# B&R Automation Studio project TD52 (part 12)

### blascompat32.h
```c
/*
 * @(#)blascompat32.h    generated by: makeheader 5.1.5  Tue May 24 21:10:38 2011
 *
 *		built from:	../../src/include/copyright.h
 *				../../src/include/pragma_interface.h
 *				include/blascompat32/blascompat32.h
 */

#if defined(_MSC_VER)
# pragma once
#endif
#if defined(__GNUC__) && (__GNUC__ > 3 || (__GNUC__ == 3 && __GNUC_MINOR__ > 3))
# pragma once
#endif

#ifndef blascompat32_h
#define blascompat32_h

/*
 * Copyright 1984-2003 The MathWorks, Inc.
 * All Rights Reserved.
 */

/* Copyright 2003-2006 The MathWorks, Inc. */

/* Only define EXTERN_C if it hasn't been defined already. This allows
 * individual modules to have more control over managing their exports.
 */
#ifndef EXTERN_C

#ifdef __cplusplus
  #define EXTERN_C extern "C"
#else
  #define EXTERN_C extern
#endif

#endif

/*
 * CONFIDENTIAL AND CONTAINING PROPRIETARY TRADE SECRETS
 * Copyright 1984-2009 The MathWorks, Inc.
 * The source code contained in this listing contains proprietary and
 * confidential trade secrets of The MathWorks, Inc.   The use, modification,
 * or development of derivative work based on the code or ideas obtained
 * from the code is prohibited without the express written permission of The
 * MathWorks, Inc.  The disclosure of this code to any party not authorized
 * by The MathWorks, Inc. is strictly forbidden.
 * CONFIDENTIAL AND CONTAINING PROPRIETARY TRADE SECRETS
 */

/*
   32-bit API wrapper for libmwblas
   WARNING: This module is a temporary module specifically designed to
            bridge the incompatiblity between Embedded MATLAB (which lacks
            a 64-bit integer type) and 64-bit BLAS only.
            Do not link to this module otherwise.
            Link to libmwblas instead.
 */
#include <tmwtypes.h>

#if defined(_WIN32)
#define FORTRAN_WRAPPER(x) x
#else
#define FORTRAN_WRAPPER(x) x ## _
#endif

#ifndef COMPLEX_TYPES
#define COMPLEX_TYPES
  typedef struct{float r,i;} complex;
  typedef struct{double r,i;} doublecomplex;
#endif

#define isamax32 FORTRAN_WRAPPER(isamax32)
EXTERN_C int isamax32(const int *n32, const float  *sx, const int *incx32);

#define idamax32 FORTRAN_WRAPPER(idamax32)
EXTERN_C int idamax32(const int *n32, const double *dx, const int *incx32);

#define icamax32 FORTRAN_WRAPPER(icamax32)
EXTERN_C int icamax32(const int *n32, const creal32_T *cx, const int *incx32);

#define izamax32 FORTRAN_WRAPPER(izamax32)
EXTERN_C int izamax32(const int *n32, const creal_T *zx, const int *incx32);

#define sasum32 FORTRAN_WRAPPER(sasum32)
EXTERN_C float sasum32(const int *n32, const float  *sx, const int *incx32);

#define dasum32 FORTRAN_WRAPPER(dasum32)
EXTERN_C double dasum32(const int *n32, const double *dx, const int *incx32);

#define saxpy32 FORTRAN_WRAPPER(saxpy32)
EXTERN_C void saxpy32(const int *n32, const float *sa, const float  *sx,
             const int *incx32, float *sy, const int *incy32);

#define daxpy32 FORTRAN_WRAPPER(daxpy32)
EXTERN_C void daxpy32(const int *n32, const double *da, const double *dx,
             const int *incx32, double *dy, const int *incy32);

#define caxpy32 FORTRAN_WRAPPER(caxpy32)
EXTERN_C void caxpy32(const int *n32, const creal32_T *ca, const creal32_T *cx,
             const int *incx32, creal32_T *cy, const int *incy32);

#define zaxpy32 FORTRAN_WRAPPER(zaxpy32)
EXTERN_C void zaxpy32(const int *n32, const creal_T *za, const creal_T *zx,
             const int *incx32, creal_T *zy, const int *incy32);

#define scopy32 FORTRAN_WRAPPER(scopy32)
EXTERN_C void scopy32(const int *n32, const float *sx, const int *incx32,
             float *sy, const int *incy32);

#define dcopy32 FORTRAN_WRAPPER(dcopy32)
EXTERN_C void dcopy32(const int *n32, const double *dx, const int *incx32,
             double *dy, const int *incy32);

#define ccopy32 FORTRAN_WRAPPER(ccopy32)
EXTERN_C void ccopy32(const int *n32, const creal32_T *cx, const int *incx32,
             creal32_T *cy, const int *incy32);

#define zcopy32 FORTRAN_WRAPPER(zcopy32)
EXTERN_C void zcopy32(const int *n32, creal_T *zx, const int *incx32,
             creal_T *zy, const int *incy32);

#define cdotc32 FORTRAN_WRAPPER(cdotc32)
EXTERN_C complex cdotc32(const int *n32, const creal32_T *cx, const int *incx32,
              const creal32_T *cy, const int *incy32);

#define zdotc32 FORTRAN_WRAPPER(zdotc32)
EXTERN_C doublecomplex zdotc32(const int *n32, const creal_T *zx, const int *incx32,
               const creal_T *zy, const int *incy32);

#define sdot32 FORTRAN_WRAPPER(sdot32)
EXTERN_C float sdot32(const int *n32, const float *sx, const int *incx32,
             const float  *sy, const int *incy32);

#define ddot32 FORTRAN_WRAPPER(ddot32)
EXTERN_C double ddot32(const int *n32, const double *dx, const int *incx32,
              const double *dy, const int *incy32);

#define cdotu32 FORTRAN_WRAPPER(cdotu32)
EXTERN_C complex cdotu32(const int *n32, const creal32_T *cx, const int *incx32,
              const creal32_T *cy, const int *incy32);

#define zdotu32 FORTRAN_WRAPPER(zdotu32)
EXTERN_C doublecomplex zdotu32(const int *n32, const creal_T *zx, const int *incx32,
               const creal_T *zy, const int *incy32);

#define sgemm32 FORTRAN_WRAPPER(sgemm32)
EXTERN_C void sgemm32(char *transa, char *transb, const int *m32, const int *n32,
             const int *k32, const float *alpha, const float *a, const int *lda32,
             const float *b, const int *ldb32, const float *beta, float *c,
             const int *ldc32);

#define dgemm32 FORTRAN_WRAPPER(dgemm32)
EXTERN_C void dgemm32(char *transa, char *transb, const int *m32, const int *n32,
             const int *k32, const double *alpha, const double *a, const int *lda32,
             const double *b, const int *ldb32, const double *beta, double  *c,
             const int *ldc32);

#define cgemm32 FORTRAN_WRAPPER(cgemm32)
EXTERN_C void cgemm32(char *transa, char *transb, const int *m32, const int *n32,
             const int *k32, const creal32_T *alpha, const creal32_T *a, const int *lda32,
             const creal32_T *b, const int *ldb32, const creal32_T *beta, creal32_T *c,
             const int *ldc32);

#define zgemm32 FORTRAN_WRAPPER(zgemm32)
EXTERN_C void zgemm32(char *transa, char *transb, const int *m32, const int *n32,
             const int *k32, const creal_T *alpha, const creal_T *a, const int *lda32,
             const creal_T *b, const int *ldb32, const creal_T *beta, creal_T *c,
             const int *ldc32);

#define sgemv32 FORTRAN_WRAPPER(sgemv32)
EXTERN_C void sgemv32(char *trans, const int *m32, const int *n32, const float *alpha,
             const float *a, const int *lda32, const float *x, const int *incx32,
             const float *beta, float *y, const int *incy32);

#define dgemv32 FORTRAN_WRAPPER(dgemv32)
EXTERN_C void dgemv32(char *trans, const int *m32, const int *n32, const double *alpha,
             const double *a, const int *lda32, const double *x, const int *incx32,
             const double *beta, double *y, const int *incy32);

#define cgemv32 FORTRAN_WRAPPER(cgemv32)
EXTERN_C void cgemv32(char *trans, const int *m32, const int *n32, const creal32_T *alpha,
             const creal32_T *a, const int *lda32, const creal32_T *x, const int *incx32,
             const creal32_T *beta, creal32_T *y, const int *incy32);

#define zgemv32 FORTRAN_WRAPPER(zgemv32)
EXTERN_C void zgemv32(char *trans, const int *m32, const int *n32, const creal_T *alpha,
             const creal_T *a, const int *lda32, const creal_T *x, const int *incx32,
             const creal_T *beta, creal_T *y, const int *incy32);

#define cgerc32 FORTRAN_WRAPPER(cgerc32)
EXTERN_C void cgerc32(const int *m32, const int *n32, const creal32_T *alpha, const creal32_T *x,
             const int *incx32, const creal32_T *y, const int *incy32,
             creal32_T *a, const int *lda32);

#define zgerc32 FORTRAN_WRAPPER(zgerc32)
EXTERN_C void zgerc32(const int *m32, const int *n32, const creal_T *alpha, const creal_T *x,
             const int *incx32, creal_T *y, const int *incy32,
             creal_T *a, const int *lda32);

#define sger32 FORTRAN_WRAPPER(sger32)
EXTERN_C void sger32(const int *m32, const int *n32, const float *alpha, const float  *x,
            const int *incx32, const float *y, const int *incy32,
            float *a, const int *lda32);

#define dger32 FORTRAN_WRAPPER(dger32)
EXTERN_C void dger32(const int *m32, const int *n32, const double *alpha, const double *x,
            const int *incx32, const double *y, const int *incy32,
            double *a, const int *lda32);

#define cgeru32 FORTRAN_WRAPPER(cgeru32)
EXTERN_C void cgeru32(const int *m32, const int *n32, const creal32_T *alpha, const creal32_T *x,
             const int *incx32, const creal32_T *y, const int *incy32,
             creal32_T *a, const int *lda32);

#define zgeru32 FORTRAN_WRAPPER(zgeru32)
EXTERN_C void zgeru32(const int *m32, const int *n32, const creal_T *alpha, const creal_T *x,
             const int *incx32, creal_T *y, const int *incy32,
             creal_T *a, const int *lda32);

#define snrm232 FORTRAN_WRAPPER(snrm232)
EXTERN_C float snrm232(const int *n32, const float *x, const int *incx32);

#define dnrm232 FORTRAN_WRAPPER(dnrm232)
EXTERN_C double dnrm232(const int *n32, const double *x, const int *incx32);

#define scnrm232 FORTRAN_WRAPPER(scnrm232)
EXTERN_C float scnrm232(const int *n32, const creal32_T *x, const int *incx32);

#define dznrm232 FORTRAN_WRAPPER(dznrm232)
EXTERN_C double dznrm232(const int *n32, const creal_T *x, const int *incx32);

#define srotg32 FORTRAN_WRAPPER(srotg32)
EXTERN_C void srotg32(float  *sa, float  *sb, float  *c, float  *s);

#define drotg32 FORTRAN_WRAPPER(drotg32)
EXTERN_C void drotg32(double *da, double *db, double *c, double *s);

#define crotg32 FORTRAN_WRAPPER(crotg32)
EXTERN_C void crotg32(creal32_T *ca, creal32_T *cb, creal32_T *c, creal32_T *s);

#define zrotg32 FORTRAN_WRAPPER(zrotg32)
EXTERN_C void zrotg32(creal_T *ca, creal_T *cb, creal_T *c, creal_T *s);

#define srot32 FORTRAN_WRAPPER(srot32)
EXTERN_C void srot32(const int *n32, float  *sx, const int *incx32, float  *sy,
            const int *incy32, const float *c, const float *s);

#define drot32 FORTRAN_WRAPPER(drot32)
EXTERN_C void drot32(const int *n32, double *dx, const int *incx32, double *dy,
            const int *incy32, const double *c, const double *s);

#define csrot32 FORTRAN_WRAPPER(csrot32)
EXTERN_C void csrot32(const int *n32, creal32_T *cx, const int *incx32, creal32_T *cy,
             const int *incy32, const float *c, const creal32_T *s);

#define zdrot32 FORTRAN_WRAPPER(zdrot32)
EXTERN_C void zdrot32(const int *n32, creal_T *cx, const int *incx32, creal_T *cy,
             const int *incy32, const double *c, const creal_T *s);

#define sscal32 FORTRAN_WRAPPER(sscal32)
EXTERN_C void sscal32(const int *n32, const float *sa, float  *sx, const int *incx32);

#define dscal32 FORTRAN_WRAPPER(dscal32)
EXTERN_C void dscal32(const int *n32, const double *da, double *dx, const int *incx32);

#define cscal32 FORTRAN_WRAPPER(cscal32)
EXTERN_C void cscal32(const int *n32, const creal32_T *ca, creal32_T *cx, const int *incx32);

#define zscal32 FORTRAN_WRAPPER(zscal32)
EXTERN_C void zscal32(const int *n32, const creal_T *za, creal_T *zx, const int *incx32);

#define sswap32 FORTRAN_WRAPPER(sswap32)
EXTERN_C void sswap32(const int *n32, float  *sx, const int *incx32, float  *sy,
             const int *incy32);

#define dswap32 FORTRAN_WRAPPER(dswap32)
EXTERN_C void dswap32(const int *n32, double *dx, const int *incx32, double *dy,
             const int *incy32);

#define cswap32 FORTRAN_WRAPPER(cswap32)
EXTERN_C void cswap32(const int *n32, creal32_T *cx, const int *incx32,
             creal32_T *cy, const int *incy32);

#define zswap32 FORTRAN_WRAPPER(zswap32)
EXTERN_C void zswap32(const int *n32, creal_T *zx, const int *incx32,
             creal_T *zy, const int *incy32);

#define strsm32 FORTRAN_WRAPPER(strsm32)
EXTERN_C void strsm32(char   *side, char   *uplo, char   *transa,
             char *diag, const int *m32, const int *n32,
             const float *alpha, const float *a, const int *lda32,
             float  *b, const int *ldb32);

#define dtrsm32 FORTRAN_WRAPPER(dtrsm32)
EXTERN_C void dtrsm32(char   *side, char   *uplo, char   *transa,
             char *diag, const int *m32, const int *n32,
             const double *alpha, const double *a, const int *lda32,
             double *b, const int *ldb32);

#define ctrsm32 FORTRAN_WRAPPER(ctrsm32)
EXTERN_C void ctrsm32(char   *side, char   *uplo, char   *transa,
             char *diag, const int *m32, const int *n32,
             const creal32_T *alpha, const creal32_T *a, const int *lda32,
             creal32_T *b, const int *ldb32);

#define ztrsm32 FORTRAN_WRAPPER(ztrsm32)
EXTERN_C void ztrsm32(char   *side, char   *uplo, char   *transa,
             char *diag, const int *m32, const int *n32,
             const creal_T *alpha, const creal_T *a, const int *lda32,
             creal_T *b, const int *ldb32);

#define strsv32 FORTRAN_WRAPPER(strsv32)
EXTERN_C void strsv32(char   *uplo, char   *trans, char   *diag,
                const int *n32, const float *a, const int *lda32,
                float *x, const int *incx32);

#define dtrsv32 FORTRAN_WRAPPER(dtrsv32)
EXTERN_C void dtrsv32(char   *uplo, char   *trans, char   *diag,
                const int *n32, const double *a, const int *lda32,
                double *x, const int *incx32);

#define ctrsv32 FORTRAN_WRAPPER(ctrsv32)
EXTERN_C void ctrsv32(char   *uplo, char   *trans, char   *diag,
                const int *n32, const creal32_T *a, const int *lda32,
                creal32_T *x, const int *incx32);

#define ztrsv32 FORTRAN_WRAPPER(ztrsv32)
EXTERN_C void ztrsv32(char   *uplo, char   *trans, char   *diag,
                const int *n32, const creal_T *a, const int *lda32,
                creal_T *x, const int *incx32);

#endif /* blascompat32_h */
```

### cg_matrx.h
```c
/* Copyright 1994-2002 The MathWorks, Inc.
 *
 * File    : cg_matrx.h      $Revision: 1.1.10.1 $ $Date: 2007/03/03 04:17:35 $
 * Abstract:
 *	Provided for backwards compatibility. See rt_matrx.h for details.
 */

#include "rt_matrx.h"

/* [EOF] cg_matrx.h */
```

### cg_sfun.h
```c
/* cg_sfun.h
 *
 * Entry point for user-written S-Functions when compiled for
 * use with the Simulink C-Code Generator.  This file should
 * be conditionally included at the bottom of any user-written
 * S-Function so as to enable the static functions within it
 * to be registered at startup.  Also, the macro S_FUNCTION_NAME
 * should be declared within the S-Function to specify the
 * entry point name--that is the name by which the S-Function
 * is to be known to the outside world.
 *
 * Copyright 1994-2005 The MathWorks, Inc.
 * $Revision: 1.15.4.9 $
 */

#ifdef __cplusplus
extern "C"
#endif

void S_FUNCTION_NAME(SimStruct *S)
{
#if S_FUNCTION_LEVEL == 1
  /* level 1 */
  ssSetmdlInitializeSizes(S, mdlInitializeSizes);
  ssSetmdlInitializeSampleTimes(S, mdlInitializeSampleTimes);
  ssSetmdlInitializeConditionsLevel1(S, mdlInitializeConditions);
  ssSetmdlOutputsLevel1(S, mdlOutputs);
  ssSetmdlUpdateLevel1(S, mdlUpdate);
  ssSetmdlDerivativesLevel1(S, mdlDerivatives);
  ssSetmdlTerminate(S, mdlTerminate);
#else
  /* user level 2 */

  ssSetmdlInitializeSizes(S, mdlInitializeSizes);
  ssSetmdlInitializeSampleTimes(S, mdlInitializeSampleTimes);

# if defined(MDL_INITIALIZE_CONDITIONS)
    ssSetmdlInitializeConditions(S, mdlInitializeConditions);
# endif
# if defined(MDL_START)
    ssSetmdlStart(S, mdlStart);
# endif

# if defined(RTW_GENERATED_ENABLE)
    ssSetRTWGeneratedEnable(S, mdlEnable);
# endif

# if defined(RTW_GENERATED_DISABLE)
    ssSetRTWGeneratedDisable(S, mdlDisable);
# endif

# if defined(MDL_ENABLE)
    ssSetmdlEnable(S, mdlEnable);
# endif

# if defined(MDL_DISABLE)
    ssSetmdlDisable(S, mdlDisable);
# endif

  ssSetmdlOutputs(S, mdlOutputs);
# if defined(MDL_GET_TIME_OF_NEXT_VAR_HIT)
    ssSetmdlGetTimeOfNextVarHit(S, mdlGetTimeOfNextVarHit);
# endif
# if defined(MDL_UPDATE)
    ssSetmdlUpdate(S, mdlUpdate);
# endif
# if defined(MDL_DERIVATIVES)
    ssSetmdlDerivatives(S, mdlDerivatives);
# endif

# if defined(MDL_PROJECTION)
    ssSetmdlProjection(S, mdlProjection);
# endif

# if defined(MDL_FORCINGFUNCTION)
    ssSetmdlForcingFunction(S, mdlForcingFunction);
# endif

# if defined(MDL_MASSMATRIX)
    ssSetmdlMassMatrix(S, mdlMassMatrix);
# endif

# if defined(MDL_RTWCG)
    ssSetmdlRTWCG(S, mdlRTWCG);
# endif

# if defined(MDL_ZERO_CROSSINGS) && (defined(MATLAB_MEX_FILE) || defined(NRT))
    ssSetmdlZeroCrossings(S, mdlZeroCrossings);
# endif

  ssSetmdlTerminate(S, mdlTerminate);
#endif
}
```

### dt_info.h
```c
/*
 * Copyright 1994-2002 The MathWorks, Inc.
 *
 * $RCSfile: dt_info.h,v $
 * $Revision: 1.17 $
 *
 * Abstract:
 *   typedef for data type transitions vectors.  Included by MODEL.dt
 */

#ifndef _DTINFO_H_
#define _DTINFO_H_

/* Data type transition */
typedef struct DataTypeTransition_tag {
  char_T *baseAddr; /* starting address of the transition  */
  int_T  dataType;
  int_T  isComplex; /* elements of this region are complex */
  int_T  nEls;
} DataTypeTransition;

/* Data type transition table */
typedef struct DataTypeTransitionTable_tag {
  uint_T             numTransitions;     /* number of transitions in table  */
  DataTypeTransition *transitions;       /* base address of transition table*/
} DataTypeTransitionTable;

/*
 * The model's data type transition info structure is attached
 * to the SimStruct:
 *
 * DataTypeTransInfo *dtInfo = ssGetModelMappingInfo(S);
 *
 * Additional information is accessed via:
 *
 * uint_T NumDataTypes     = dtGetNumDataTypes(dtInfo);
 * uint_T DataTypeSizes[]  = dtGetDataTypeSizes(dtInfo);
 * char_T *DataTypeNames[] = dtGetDataTypeNames(dtInfo);
 *
 * DataTypeTransTable *B     = dtGetBIODataTypeTrans(dtInfo);
 * DataTypeTransTable *P     = dtGetParamDataTypeTrans(dtInfo);
 * DataTypeTransTable *DWork = dtGetDWorkDataTypeTrans(dtInfo);
 * DataTypeTransTable *Xd    = dtGetDiscStatesDataTypeTrans(dtInfo);
 * DataTypeTransTable *U     = dtGetExternalInputsDataTypeTrans(dtInfo);
 * DataTypeTransTable *Y     = dtGetExternalOutputsDataTypeTrans(dtInfo);
 *
 * And, using the block outputs as an example
 *
 * uint_T              NumBIOTransitions  = dtGetNumTransitions(B);
 * DataTypeTransition  *BIOTransitions    = dtGetTransitions(B);
 * char_T              *address           = dtTransGetAddress(B, idx);
 * int_T               dataType           = dtTransGetDataType(B, idx);
 * int_T               isComplex          = dtTransGetComplexFlag(B, idx);
 *
 * where, idx is the index into the block outputs transition table.
 * For example, dtTransGetComplexFlag(B, 5) indicates whether the fifth
 * transition represents a complex region of the block outputs structure
 * structure and dtTransGetAddress(B, 5) is the absolute base address of
 * the region.
 */

typedef struct DataTypeTransInfo_tag {
  uint_T         numDataTypes;    /* number of data types in model    */
  uint_T         *dataTypeSizes;  /* data types (bytes) of data types */
  char_T  const **dataTypeNames;  /* names of data types              */

  DataTypeTransitionTable *B;      /* block outputs */
  DataTypeTransitionTable *P;      /* parameters */
  DataTypeTransitionTable *DWork;  /* data type work vector */
  DataTypeTransitionTable *Xd;     /* discrete states */
  DataTypeTransitionTable *U;      /* model inputs */
  DataTypeTransitionTable *Y;      /* model outputs */
} DataTypeTransInfo;

#define dtGetNumDataTypes(dtInfo)   ((uint_T)((dtInfo)->numDataTypes))
#define dtGetDataTypeSizes(dtInfo)  ((dtInfo)->dataTypeSizes)
#define dtGetDataTypeNames(dtInfo)  ((dtInfo)->dataTypeNames)

#define dtGetBIODataTypeTrans(dtInfo)             ((dtInfo)->B)
#define dtGetParamDataTypeTrans(dtInfo)           ((dtInfo)->P)
#define dtGetDWorkDataTypeTrans(dtInfo)           ((dtInfo)->DWork)
#define dtGetDiscStatesDataTypeTrans(dtInfo)      ((dtInfo)->Xd)
#define dtGetExternalInputsDataTypeTrans(dtInfo)  ((dtInfo)->U)
#define dtGetExternalOutputsDataTypeTrans(dtInfo) ((dtInfo)->Y)

#define dtGetNumTransitions(dtTable) \
    ((dtTable)->numTransitions)

#define dtGetTransitions(dtTable) \
    ((dtTable)->transitions)

#define dtTransGetAddress(dtTable, idx) \
    ((dtTable)->transitions[(idx)].baseAddr)

#define dtTransGetDataType(dtTable, idx) \
    ((dtTable)->transitions[(idx)].dataType)

#define dtTransNEls(dtTable, idx) \
    ((dtTable)->transitions[(idx)].nEls)

#define dtTransGetComplexFlag(dtTable, idx) \
    ((dtTable)->transitions[(idx)].isComplex)

#endif /* _DTINFO_ */
```

### emlrt.h
```c
/*
 * @(#)emlrt.h    generated by: makeheader 5.1.5  Tue May 24 21:21:44 2011
 *
 *		built from:	../../../src/include/copyright.h
 *				../../../src/include/pragma_interface.h
 *				AAContext.cpp
 *				Alias.cpp
 *				AllocCheck.cpp
 *				Assign.cpp
 *				BoundsCheck.cpp
 *				Create.cpp
 *				CreateArray.cpp
 *				Destroy.cpp
 *				Display.cpp
 *				DoubleCheck.cpp
 *				ExternalMode.cpp
 *				Gateway.cpp
 *				HeapMemoryCheck.cpp
 *				HeapReferenceStack.cpp
 *				InitArray.cpp
 *				Logging.cpp
 *				MultipleEntryPoints.cpp
 *				ParallelMode.cpp
 *				RefCount.cpp
 *				RunTimeErrors.cpp
 *				RunTimeLocationLogging.cpp
 *				RunTimeStack.cpp
 *				Serialize.cpp
 *				Signals.cpp
 *				SizeEqCheck.cpp
 *				TypeCheck.cpp
 *				VSArray.cpp
 */

#if defined(_MSC_VER)
# pragma once
#endif
#if defined(__GNUC__) && (__GNUC__ > 3 || (__GNUC__ == 3 && __GNUC_MINOR__ > 3))
# pragma once
#endif

#ifndef emlrt_h
#define emlrt_h

/*
 * Copyright 1984-2003 The MathWorks, Inc.
 * All Rights Reserved.
 */

/* Copyright 2003-2006 The MathWorks, Inc. */

/* Only define EXTERN_C if it hasn't been defined already. This allows
 * individual modules to have more control over managing their exports.
 */
#ifndef EXTERN_C

#ifdef __cplusplus
  #define EXTERN_C extern "C"
#else
  #define EXTERN_C extern
#endif

#endif

/*
 * MATLAB INTERNAL USE ONLY :: MEX Version
 */
#define EMLRT_VERSION_R2010B 0x2010B
#define EMLRT_VERSION_R2011A 0x2011A
#define EMLRT_VERSION_R2011B 0x2011B
#define EMLRT_VERSION_INFO  EMLRT_VERSION_R2011B

/*
 * MATLAB INTERNAL USE ONLY :: MEX error function
 */
typedef void (*EmlrtErrorFunction)(const char* aIdentifier, const CHAR16_T* aMessage, int32_T aTId);

/*
 * MATLAB INTERNAL USE ONLY :: Prototype of free functions.
 */
typedef void (*EmlrtHeapReferenceFreeFcn)(void *, boolean_T);

/*
 * MATLAB INTERNAL USE ONLY :: Runtime message identifier
 */
typedef struct emlrtMsgIdentifier {
    const char *fIdentifier;
    const struct emlrtMsgIdentifier *fParent;
} emlrtMsgIdentifier;

/*
 * MATLAB INTERNAL USE ONLY :: Runtime stack info
 */
typedef struct emlrtRSInfo {
    int32_T     lineNo;
    const char *fcnName;
    const char *pathName;
} emlrtRSInfo;

/*
 * MATLAB INTERNAL USE ONLY :: Runtime call stack
 */
typedef struct emlrtCallStack {
    uint32_T*    fRTStackPointer;       /* expanded by numCores */
    uint32_T*    fRTStackSize;          /* expanded by numCores */
    const emlrtRSInfo*** fRTStackInfo;  /* expanded by numCores */
    struct emlrtContext *fRTContext;
    uint32_T     fRTStackBranch;
} emlrtCallStack;

/*
 * MATLAB INTERNAL USE ONLY :: MEX Context
 */
typedef struct emlrtContext {
    boolean_T   bFirstTime;
    boolean_T   bInitialized;
    unsigned int fVersionInfo;
    EmlrtErrorFunction fErrorFunction;
    const char *fFunctionName;
    struct emlrtCallStack* fRTCallStack;
    boolean_T   bDebugMode;
    void *fLoggingContext;
    boolean_T bParallelMode;
    int32_T                fNumCores;
    void *fLocationLoggingContext;
    boolean_T bWarningInsideParallelRegion;
} emlrtContext;

/*
 * MATLAB INTERNAL USE ONLY :: External Mode Simulation
 */
typedef struct emlrtExternalSim {
    void        *fESim;
    uint8_T     *fIOBuffer;
    uint8_T     *fIOBufHead;
    size_t       fIOBufSize;
} emlrtExternalSim;

/*
 * MATLAB INTERNAL USE ONLY :: Array bounds check parameters
 */
typedef struct emlrtBCInfo {
    int32_T     iFirst;
    int32_T     iLast;
    int32_T     lineNo;
    int32_T     colNo;
    const char *aName;
    const char *fName;
    const char *pName;
    int32_T     checkKind; /* see src/cg_ir/classic/cg_node.hpp::CG_BoundsCheckKindEnum */
}   emlrtBCInfo;

/*
 * MATLAB INTERNAL USE ONLY :: Equality check parameters
 */
typedef struct emlrtECInfo {
    int32_T     nDims;
    int32_T     lineNo;
    int32_T     colNo;
    const char *fName;
    const char *pName;
}   emlrtECInfo;

/*
 * MATLAB INTERNAL USE ONLY :: Array bounds check parameters
 */
typedef struct {
    int32_T     lineNo;
    int32_T     colNo;
    const char *fName;
    const char *pName;
}   emlrtRTEInfo;

typedef emlrtRTEInfo emlrtMCInfo;

/* MATLAB INTERNAL USE ONLY :: Reference to global runtime context */
extern emlrtContext emlrtContextGlobal;

/*
 * MATLAB INTERNAL USE ONLY :: Initialize run-time context
 */
EXTERN_C void
emlrtInitContext(struct emlrtContext *ctx);

/*
 * MATLAB INTERNAL USE ONLY :: Query first-time sentinel
 */
EXTERN_C boolean_T
emlrtFirstTime(struct emlrtContext *aMAInfo);

/*
 * MATLAB INTERNAL USE ONLY :: Exit Time Cleanup
 */
EXTERN_C void
emlrtExitTimeCleanup(struct emlrtContext *aMAInfo);

/*
 * MATLAB INTERNAL USE ONLY :: Create an mxArray alias
 */
EXTERN_C const mxArray *
emlrtAlias(const mxArray *in);

/*
 * MATLAB INTERNAL USE ONLY :: Create a persistent mxArray alias
 */
EXTERN_C const mxArray *
emlrtAliasP(const mxArray *in);

/*
 * MATLAB INTERNAL USE ONLY :: Create an mxArray vector alias
 */
EXTERN_C void
emlrtAliases(int32_T nlhs, const mxArray **plhs, const mxArray **prhs);

/*
 * MATLAB INTERNAL USE ONLY :: Return an mxArray to MATLAB
 */
EXTERN_C mxArray *
emlrtReturnArrayR2009a(const mxArray *pa);

/*
 * MATLAB INTERNAL USE ONLY :: Simulation hysteresis suppression
 */
EXTERN_C void
emlrtShs(const void *a, const int b);

/*
 * MATLAB INTERNAL USE ONLY :: Verify default fimath
 */
EXTERN_C void
emlrtCheckDefaultFimathR2008b(const mxArray **ctFimath);

/*
 * MATLAB INTERNAL USE ONLY :: Clear mxArray allocation count
 */
EXTERN_C void
emlrtClearAllocCount(struct emlrtContext *aMAInfo, boolean_T bM, uint32_T iL, const char* ctDTO);

/*
 * MATLAB INTERNAL USE ONLY :: Update mxArray allocation count
 */
EXTERN_C void
emlrtUpdateAllocCount(int32_T delta);

/*
 * MATLAB INTERNAL USE ONLY :: Update persistent mxArray allocation count
 */
EXTERN_C void
emlrtUpdateAllocCountP(int32_T delta);

/*
 * MATLAB INTERNAL USE ONLY :: Check mxArray allocation count
 */
EXTERN_C void
emlrtCheckAllocCount(void);

/*
 * MATLAB INTERNAL USE ONLY :: Assign to an mxArray
 */
EXTERN_C void
emlrtAssign(const mxArray **lhs, const mxArray *rhs);

/*
 * MATLAB INTERNAL USE ONLY :: Assign to a persistent mxArray
 */
EXTERN_C void
emlrtAssignP(const mxArray **lhs, const mxArray *rhs);

/*
 * MATLAB INTERNAL USE ONLY :: Assign to a vector of mxArrays
 */
EXTERN_C void
emlrtAssigns(int32_T nlhs, const mxArray **plhs, const mxArray **prhs);

/*
 * MATLAB INTERNAL USE ONLY :: Array bounds check
 */
EXTERN_C int32_T
emlrtBoundsCheck(int32_T indexValue, emlrtBCInfo *aInfo);

/*
 * MATLAB INTERNAL USE ONLY :: Array bounds check
 */
EXTERN_C int32_T
emlrtBoundsCheckR2011a(int32_T indexValue, emlrtBCInfo *aInfo, struct emlrtContext *aContext);

/*
 * MATLAB INTERNAL USE ONLY :: Array bounds check
 */
EXTERN_C int32_T
emlrtBoundsCheckR2011b(int32_T indexValue, emlrtBCInfo *aInfo, struct emlrtContext *aContext, int32_T aTId);

/*
 * MATLAB INTERNAL USE ONLY :: Dynamic array bounds check
 */
EXTERN_C int32_T
emlrtDynamicBoundsCheck(int32_T indexValue, int32_T loBound, int32_T hiBound, emlrtBCInfo *aInfo);

/*
 * MATLAB INTERNAL USE ONLY :: Dynamic array bounds check
 */
EXTERN_C int32_T
emlrtDynamicBoundsCheckR2011a(int32_T indexValue, int32_T loBound, int32_T hiBound, emlrtBCInfo *aInfo, struct emlrtContext *aContext);

/*
 * MATLAB INTERNAL USE ONLY :: Dynamic array bounds check
 */
EXTERN_C int32_T
emlrtDynamicBoundsCheckR2011b(int32_T indexValue, int32_T loBound, int32_T hiBound, emlrtBCInfo *aInfo, struct emlrtContext *aContext, int32_T aTId);

/*
 * MATLAB INTERNAL USE ONLY :: Perform integer multiplication, raise runtime error
 *                             if the operation overflows.
 */
EXTERN_C size_t emlrtSizeMul(size_t s1, size_t s2, const emlrtRTEInfo *aInfo);

/*
 * MATLAB INTERNAL USE ONLY :: Perform integer multiplication, raise runtime error
 *                             if the operation overflows.
 */
EXTERN_C size_t emlrtSizeMulR2011b(size_t s1, size_t s2, const emlrtRTEInfo *aInfo, struct emlrtContext *aContext, int32_T aTId);

/*
 * MATLAB INTERNAL USE ONLY :: Create an mxArray string from a C string
 */
EXTERN_C const mxArray *
emlrtCreateString(const char *in);

/*
 * MATLAB INTERNAL USE ONLY :: Create an mxArray string from a single char
 */
EXTERN_C const mxArray *
emlrtCreateString1(char c);

/*
 * MATLAB INTERNAL USE ONLY :: Create a struct matrix mxArray
 */
EXTERN_C const mxArray *
emlrtCreateStructMatrix(int32_T m, int32_T n, int32_T nfields, const char **field_names);

/*
 * MATLAB INTERNAL USE ONLY :: Create a struct matrix mxArray
 */
EXTERN_C const mxArray *
emlrtCreateStructArray(int32_T ndim, const int32_T *pdim, int32_T nfields, const char **field_names);

/*
 * MATLAB INTERNAL USE ONLY :: Create an enum
 */
EXTERN_C const mxArray *
emlrtCreateEnumR2010a(struct emlrtContext *ctx, const char *name, const mxArray *data);

/*
 * MATLAB INTERNAL USE ONLY :: Create an enum
 */
EXTERN_C const mxArray *
emlrtCreateEnumR2009a(const char *name, const mxArray *data);

/*
 * MATLAB INTERNAL USE ONLY :: Add a field to a struct matrix mxArray
 */
EXTERN_C const mxArray *
emlrtAddField(const mxArray *mxStruct, const mxArray *mxField, const char *fldName, int index);

/*
 * MATLAB INTERNAL USE ONLY :: Get a field from a struct matrix mxArray
 */
EXTERN_C const mxArray *
emlrtGetField(const mxArray *mxStruct, int aIndex, const char *fldName);

/*
 * MATLAB INTERNAL USE ONLY :: Create a numeric matrix mxArray
 */
EXTERN_C const mxArray *
emlrtCreateNumericMatrix(int32_T m, int32_T n, int32_T classID, int32_T nComplexFlag);

/*
 * MATLAB INTERNAL USE ONLY :: Create a numeric matrix mxArray
 */
EXTERN_C const mxArray *
emlrtCreateNumericArray(int32_T ndim, const void *pdim, int32_T classID, int32_T nComplexFlag);

/*
 * MATLAB INTERNAL USE ONLY :: Create a scaled numeric matrix mxArray
 */
EXTERN_C const mxArray *
emlrtCreateScaledNumericArrayR2008b(int32_T ndim, const void *pdim, int32_T classID, int32_T nComplexFlag, int32_T aScale);

/*
 * MATLAB INTERNAL USE ONLY :: Create a double scalar mxArray
 */
EXTERN_C const mxArray *
emlrtCreateDoubleScalar(real_T in);

/*
 * MATLAB INTERNAL USE ONLY :: Create a logical matrix mxArray
 */
EXTERN_C const mxArray *
emlrtCreateLogicalMatrix(int32_T m, int32_T n);

/*
 * MATLAB INTERNAL USE ONLY :: Create a logical matrix mxArray
 */
EXTERN_C const mxArray *
emlrtCreateLogicalArray(int32_T ndim, const int32_T *dims);

/*
 * MATLAB INTERNAL USE ONLY :: Create a logical scalar mxArray
 */
EXTERN_C const mxArray *
emlrtCreateLogicalScalar(boolean_T in);

/*
 * MATLAB INTERNAL USE ONLY :: Create a character array mxArray
 */
EXTERN_C const mxArray *
emlrtCreateCharArray(int32_T ndim, const int32_T *dims);

/*
 * MATLAB INTERNAL USE ONLY :: Create a 2-D character array mxArray
 */
EXTERN_C const mxArray *
emlrtCreateCharArray2(int32_T m, int32_T n);

/*
 * MATLAB INTERNAL USE ONLY :: Create a numerictype mxArray
 */
EXTERN_C const mxArray *
 emlrtCreateNumericType(boolean_T issigned, int32_T wordlength, real_T bias, real_T slope, int32_T fixedexponent);

/*
 * MATLAB INTERNAL USE ONLY :: Create a FI mxArray from a value mxArray
 */
EXTERN_C const mxArray *emlrtCreateFI(const mxArray *fimath, const mxArray *ntype, const char *fitype, const mxArray *fival);

/*
 * MATLAB INTERNAL USE ONLY :: Create a FI mxArray from a value mxArray
 */
EXTERN_C const mxArray *emlrtCreateFIR2009a(const mxArray *fimath, const mxArray *ntype, const char *fitype, const mxArray *fival, const bool fmIsLocal);

/*
 * MATLAB INTERNAL USE ONLY :: Get the intarray from a FI mxArray
 */
EXTERN_C const mxArray *emlrtImportFiIntArrayR2008b(const mxArray *aFiMx);

/*
 * MATLAB INTERNAL USE ONLY :: Get the enum int from an MCOS enumeration mxArray.
 */
EXTERN_C const int32_T emlrtGetEnumElementR2009a(const mxArray *aEnum, int aIndex);

/*
 * MATLAB INTERNAL USE ONLY :: Get the enum int from an MCOS enumeration mxArray.
 */
EXTERN_C const mxArray * emlrtGetEnumUnderlyingArrayR2009a(const mxArray *aEnum);

/*
 * MATLAB INTERNAL USE ONLY :: Create an array of mxArrays
 */
EXTERN_C const mxArray *
emlrtCreateArray(const mxArray **ppa, int_T am, int_T an);

/*
 * MATLAB INTERNAL USE ONLY :: Destroy an mxArray
 */
EXTERN_C void
emlrtDestroyArray(const mxArray **pa);

/*
 * MATLAB INTERNAL USE ONLY :: Destroy a vector of mxArrays
 */
EXTERN_C void
emlrtDestroyArrays(int32_T narrays, const mxArray **parrays);

/*
 * MATLAB INTERNAL USE ONLY :: Display an mxArray
 */
EXTERN_C void
emlrtDisplayR2011a(const mxArray *pa, const char *name);

/*
 * MATLAB INTERNAL USE ONLY :: Display an mxArray
 */
EXTERN_C void
emlrtDisplayR2011b(const mxArray *pa, const char *name, emlrtMCInfo* aLoc, int32_T aTId);

/*
 * MATLAB INTERNAL USE ONLY :: Double check parameters
 */
typedef struct {
    int32_T     lineNo;
    int32_T     colNo;
    const char *fName;
    const char *pName;
    int32_T     checkKind; /* see src/cg_ir/classic/cg_node.hpp::CG_Node_CheckEnum */
}   emlrtDCInfo;

/*
 * MATLAB INTERNAL USE ONLY :: Check that d can be safely cast to int.
 */
EXTERN_C real_T
emlrtIntegerCheckR2009b(real_T d, emlrtDCInfo *aInfo);

/*
 * MATLAB INTERNAL USE ONLY :: Check that d can be safely cast to int.
 */
EXTERN_C real_T
emlrtIntegerCheckR2011a(real_T d, emlrtDCInfo *aInfo, struct emlrtContext *aContext);

/*
 * MATLAB INTERNAL USE ONLY :: Check that d can be safely cast to int.
 */
EXTERN_C real_T
emlrtIntegerCheckR2011b(real_T d, emlrtDCInfo *aInfo, struct emlrtContext *aContext, int32_T aTId);

/*
 * MATLAB INTERNAL USE ONLY :: Check that d is not NaN.
 */
EXTERN_C real_T
emlrtNotNanCheckR2009b(real_T d, emlrtDCInfo *aInfo);

/*
 * MATLAB INTERNAL USE ONLY :: Check that d is not NaN.
 */
EXTERN_C real_T
emlrtNotNanCheckR2011a(real_T d, emlrtDCInfo *aInfo, struct emlrtContext *aContext);

/*
 * MATLAB INTERNAL USE ONLY :: Check that d is not NaN.
 */
EXTERN_C real_T
emlrtNotNanCheckR2011b(real_T d, emlrtDCInfo *aInfo, struct emlrtContext *aContext, int32_T aTId);

/*
 * MATLAB INTERNAL USE ONLY :: Check that d >= 0.
 */
EXTERN_C real_T
emlrtNonNegativeCheckR2009b(real_T d, emlrtDCInfo *aInfo);

/*
 * MATLAB INTERNAL USE ONLY :: Check that d >= 0.
 */
EXTERN_C real_T
emlrtNonNegativeCheckR2011a(real_T d, emlrtDCInfo *aInfo, struct emlrtContext *aContext);

/*
 * MATLAB INTERNAL USE ONLY :: Check that d >= 0.
 */
EXTERN_C real_T
emlrtNonNegativeCheckR2011b(real_T d, emlrtDCInfo *aInfo, struct emlrtContext *aContext, int32_T aTId);

/*
 * MATLAB INTERNAL USE ONLY :: Check that the loop has an integer number of iterations.
 */
EXTERN_C boolean_T
emlrtForLoopVectorIsValidR2011b(real_T start, real_T step, real_T end, mxClassID classID, int n);

/*
 * MATLAB INTERNAL USE ONLY :: Check that the loop has an integer number of iterations.
 */
EXTERN_C void
emlrtForLoopVectorCheckR2011b(real_T start, real_T step, real_T end, mxClassID classID, int n, emlrtRTEInfo *aInfo, struct emlrtContext *aContext, int32_T aTId);

#ifdef __WATCOMC__
#pragma aux emlrtIntegerCheckR2009b value [8087];
#pragma aux emlrtNotNanCheckR2009b value [8087];
#pragma aux emlrtNonNegativeCheckR2009b value [8087];
#pragma aux emlrtIntegerCheckR2011a value [8087];
#pragma aux emlrtNotNanCheckR2011a value [8087];
#pragma aux emlrtNonNegativeCheckR2011a value [8087];
#pragma aux emlrtIntegerCheckR2011b value [8087];
#pragma aux emlrtNotNanCheckR2011b value [8087];
#pragma aux emlrtNonNegativeCheckR2011b value [8087];
#endif

/*
 * MATLAB INTERNAL USE ONLY :: Terminate external-mode serialization
 */
EXTERN_C void
emlrtExtSerializeEnd(struct emlrtExternalSim *aExternalSim);

/*
 * MATLAB INTERNAL USE ONLY :: Deserialize a byte
 */
EXTERN_C uint8_T
emlrtExtDeserializeByte(struct emlrtExternalSim *aExternalSim);

/*
 * MATLAB INTERNAL USE ONLY :: Serialize a byte
 */
EXTERN_C void
emlrtExtSerializeByte(struct emlrtExternalSim *aExternalSim, uint8_T b);

/*
 * MATLAB INTERNAL USE ONLY :: Deserialize a single
 */
EXTERN_C real32_T
emlrtExtDeserializeSingle(struct emlrtExternalSim *aExternalSim);

/*
 * MATLAB INTERNAL USE ONLY :: Serialize a single
 */
EXTERN_C void
emlrtExtSerializeSingle(struct emlrtExternalSim *aExternalSim, real32_T s);

/*
 * MATLAB INTERNAL USE ONLY :: Deserialize a double
 */
EXTERN_C real64_T
emlrtExtDeserializeDouble(struct emlrtExternalSim *aExternalSim);

/*
 * MATLAB INTERNAL USE ONLY :: Serialize a double
 */
EXTERN_C void
emlrtExtSerializeDouble(struct emlrtExternalSim *aExternalSim, real64_T d);

/*
* MATLAB INTERNAL USE ONLY :: connect to external target
*/
EXTERN_C void
emlrtExtConnect(struct emlrtExternalSim *aExternalSim, const uint32_T aChecksum[4], const char *aMexArgs, const char *aMethod);

/*
* MATLAB INTERNAL USE ONLY :: disconnect from external target
*/
EXTERN_C void
emlrtExtDisconnect(struct emlrtExternalSim *aExternalSim);

#ifdef __WATCOMC__
#pragma aux emlrtExtDeserializeDouble value [8087];
#endif

/*
* MATLAB INTERNAL USE ONLY :: fetch a global variable
*/
EXTERN_C void
emlrtPutGlobalVariable(const char *name, const mxArray *parray);

/*
* MATLAB INTERNAL USE ONLY :: fetch a global variable
*/
EXTERN_C const mxArray *
emlrtGetGlobalVariable(const char *name);

/*
 * MATLAB INTERNAL USE ONLY :: Call out to MATLAB
 */
EXTERN_C const mxArray *
emlrtCallMATLAB(int32_T nlhs, const mxArray **plhs, int32_T nrhs, const mxArray **prhs, const char *cmd, boolean_T tmp, emlrtMCInfo* aLoc);

/*
 * MATLAB INTERNAL USE ONLY :: Call out to MATLAB
 */
EXTERN_C const mxArray *
emlrtCallMATLABR2011b(int32_T nlhs, const mxArray **plhs, int32_T nrhs, const mxArray **prhs, const char *cmd, boolean_T tmp, emlrtMCInfo* aLoc, struct emlrtContext *aContext, int32_T aTId);

/*
 * MATLAB INTERNAL USE ONLY :: Maintain heap memory check information upon entering a mex function.
 */
EXTERN_C void emlrtHeapMemCheckInitialize(struct emlrtContext *aMexContext, int aMaxHeapSize);

/*
 * MATLAB INTERNAL USE ONLY :: Maintain heap memory check information upon leaving a mex function.
 */
EXTERN_C void emlrtHeapMemCheckTerminate(void);

/*
 * MATLAB INTERNAL USE ONLY :: Register the mex function to be unloaded.
 */
EXTERN_C void emlrtHeapMemCheckPrepareUnload(emlrtContext *aMexContext);

/*
 * MATLAB INTERNAL USE ONLY :: Maintain heap memory check information upon unload a mex function.
 *                             Memory leak check is performed at this moment no matter for normal or error exit.
 */
EXTERN_C void emlrtHeapMemCheckUnloadMex(struct emlrtContext *aMexContext);

/*
 * MATLAB INTERNAL USE ONLY :: malloc with memory integrity check
 */
EXTERN_C void* emlrtMalloc(size_t aSize);

/*
 * MATLAB INTERNAL USE ONLY :: calloc with memory integrity check
 */
EXTERN_C void* emlrtCalloc(size_t aNum, size_t aSize);

/*
 * MATLAB INTERNAL USE ONLY :: free with memory integrity check
 */
EXTERN_C void emlrtFree(void *aPtr);

/*
 * MATLAB INTERNAL USE ONLY :: Enter a new function of a MEX call.
 */
EXTERN_C void emlrtHeapReferenceStackEnterFcn(void);

/*
 * MATLAB INTERNAL USE ONLY :: Enter a new function of a MEX call.
 */
EXTERN_C void emlrtHeapReferenceStackLeaveFcn(void);

/*
 * MATLAB INTERNAL USE ONLY :: Push a new entry to the heap reference stack.
 */
EXTERN_C void emlrtPushHeapReferenceStack(void *aHeapReference, EmlrtHeapReferenceFreeFcn aFreeFcn);

/*
 * MATLAB INTERNAL USE ONLY :: Initialize a character mxArray
 */
EXTERN_C void
emlrtInitCharArray(int32_T n, const mxArray *a, const char *s);

/*
 * MATLAB INTERNAL USE ONLY :: Initialize a logical mxArray
 */
EXTERN_C void
emlrtInitLogicalArray(int32_T n, const mxArray *a, const boolean_T *b);

/*
 * MATLAB INTERNAL USE ONLY :: Export a numeric mxArray
 */
EXTERN_C void
emlrtExportNumericArrayR2008b(const mxArray *aOut, const void *aInData, int32_T aElementSize);

#define EMLRT_LOGGING_UPDATE_RANGE(v1,v2,v3)                                          \
{                                                                                     \
    static void* range = 0;                                                           \
    if (range == 0) {                                                                 \
        range = emlrtLoggingContextGetRangeInfo(&emlrtContextGlobal,(v1),(v2), (v3)); \
    } else {                                                                          \
        emlrtLoggingContextUpdateRangeInfo(range, (v3));                              \
    }                                                                                 \
}

/*
* MATLAB INTERNAL USE ONLY :: Log Range
*/

EXTERN_C void* emlrtLoggingContextGetRangeInfo(struct emlrtContext *aMAInfo, const char *aFunctionName, const char *aExprName, double defaultValue);

/*
* MATLAB INTERNAL USE ONLY :: Log Range
*/

EXTERN_C void emlrtLoggingContextUpdateRangeInfo(void* rangeInfo, double aValue);

/*
* MATLAB INTERNAL USE ONLY :: Marshall Logging Info to MATLAB
*/

EXTERN_C mxArray* emlrtLoggingContextToMxArray(struct emlrtContext *aMAInfo);

/*
 * MATLAB INTERNAL USE ONLY :: Auto-generated mexFunction
 */
typedef void (*emlrtMexFunction)(int, mxArray*[], int, const mxArray*[]);
/*
 * MATLAB INTERNAL USE ONLY :: Auto-generated entry-point
 */
typedef struct emlrtEntryPoint {
    const char *fName;
    emlrtMexFunction fMethod;
} emlrtEntryPoint;

/*
 * MATLAB INTERNAL USE ONLY :: Lookup an entry point
 */
EXTERN_C emlrtMexFunction
emlrtGetMethod(int nrhs, const mxArray *prhs[], struct emlrtEntryPoint *aEntryPoints, int aNumEntryPoints);

#define EMLRTENTERPARALLELREGION() { \
    emlrtContextGlobal.fRTCallStack->fRTStackBranch = emlrtContextGlobal.fRTCallStack->fRTStackPointer[0];  \
    emlrtContextGlobal.bWarningInsideParallelRegion = false;      \
    emlrtContextGlobal.bParallelMode = true;                      \
}

#define EMLRTEXITPARALLELREGION(iserror) { \
    emlrtContextGlobal.bParallelMode = false;                     \
    if (iserror){                                                 \
        emlrtHandleParallelRunTimeError();                        \
    }                                                             \
    if (emlrtContextGlobal.bWarningInsideParallelRegion) {        \
        emlrtHandleParallelSuppressedWarning();                   \
    }                                                             \
    emlrtContextGlobal.fRTCallStack->fRTStackBranch = 0;          \
}

/*
 * MATLAB INTERNAL USE ONLY :: Check that d can be safely cast to int.
 */
EXTERN_C bool
emlrtIsMATLABThread(int32_T aTId);

/*
 * MATLAB INTERNAL USE ONLY :: Check that d can be safely cast to int.
 */
EXTERN_C bool
emlrtSetWarningFlag(struct emlrtContext *aContext, int32_T aTId);

/*
 * MATLAB INTERNAL USE ONLY :: Create a shallow copy of an mxArray
 */
EXTERN_C const mxArray *
emlrtCreateReference(const mxArray *pa);

/*
 * MATLAB INTERNAL USE ONLY :: Division by zero error
 */
EXTERN_C void
emlrtDivisionByZeroError(void);

/*
 * MATLAB INTERNAL USE ONLY :: Division by zero error
 */
EXTERN_C void
emlrtDivisionByZeroErrorR2008a(const emlrtRTEInfo *aInfo);

/*
 * MATLAB INTERNAL USE ONLY :: Division by zero error
 */
EXTERN_C void
emlrtDivisionByZeroErrorR2011b(const emlrtRTEInfo *aInfo, struct emlrtContext *aContext, int32_T aTId);

/*
 * MATLAB INTERNAL USE ONLY :: Integer overflow error
 */
EXTERN_C void
emlrtIntegerOverflowErrorR2008a(const emlrtRTEInfo *aInfo);

/*
 * MATLAB INTERNAL USE ONLY :: Integer overflow error
 */
EXTERN_C void
emlrtIntegerOverflowErrorR2011b(const emlrtRTEInfo *aInfo, struct emlrtContext *aContext, int32_T aTId);

/*
 * MATLAB INTERNAL USE ONLY :: Raise C heap allocation failure
 */
EXTERN_C void emlrtHeapAllocationError(const emlrtRTEInfo *aInfo);

/*
 * MATLAB INTERNAL USE ONLY :: Raise C heap allocation failure
 */
EXTERN_C void emlrtHeapAllocationErrorR2011b(const emlrtRTEInfo *aInfo, struct emlrtContext *aContext, int32_T aTId);

/*
 * MATLAB INTERNAL USE ONLY :: Error with given message ID.
 */
EXTERN_C void emlrtErrorWithMessageID(const char* aMsgID, const emlrtRTEInfo *aInfo);

/*
 * MATLAB INTERNAL USE ONLY :: Error with given message ID.
 */
EXTERN_C void emlrtErrorWithMessageIDR2011b(const char* aMsgID, const emlrtRTEInfo *aInfo, struct emlrtContext *aContext, int32_T aTId);

/*
 * MATLAB INTERNAL USE ONLY :: Convert a message ID to a heap-allocated LCP string.
 * This function is used by Stateflow run-time library only.
 */
EXTERN_C char* emlrtTranslateMessageIDtoLCPstring(const char* aMsgID);

/*
 * MATLAB INTERNAL USE ONLY :: Convert a UTF16 message string to a heap-allocated LCP string.
 * This function is used by Stateflow run-time library only.
 */
EXTERN_C char* emlrtTranslateUTF16MessagetoLCPstring(const CHAR16_T* aUTF16Msg);

typedef struct
{
    char * MexFileName;
    char * TimeStamp;
    char * buildDir;
    int32_T numFcns;
} emlrtLocationLoggingFileInfoType;

typedef struct
{
    char * FunctionName;
    int32_T FunctionID;
    int32_T numInstrPoints;
} emlrtLocationLoggingFunctionInfoType;

typedef struct
{
    real_T SimMin;
    real_T SimMax;
    int32_T OverflowWraps;
    int32_T Saturations;
    boolean_T IsAlwaysInteger;
} emlrtLocationLoggingDataType;

typedef struct
{
    int32_T MxInfoID;
    int32_T TextStart;
    int32_T TextLength;
    int16_T Reason;
    boolean_T MoreLocations;
} emlrtLocationLoggingLocationType;

/*
 * MATLAB INTERNAL USE ONLY :: Get LocationLogging Info
 */
EXTERN_C mxArray* emlrtLocationLoggingPullLog(const char* const MexFileName);

/*
 * MATLAB INTERNAL USE ONLY :: Save LocationLogging Info
 */
EXTERN_C void emlrtLocationLoggingPushLog(const emlrtLocationLoggingFileInfoType* const fileInfo,
                                 const emlrtLocationLoggingFunctionInfoType* const functionInfoTable,
                                 const emlrtLocationLoggingDataType* const dataTables,
                                 const emlrtLocationLoggingLocationType* const locationTables
    );

/*
 * MATLAB INTERNAL USE ONLY :: Clear LocationLogging Info
 */
EXTERN_C bool emlrtLocationLoggingClearLog(const char* const MexFileName);

/*
 * MATLAB INTERNAL USE ONLY :: List entries in LocationLogging Info
 */
EXTERN_C mxArray* emlrtLocationLoggingListLogs(void);

/*
 * MATLAB INTERNAL USE ONLY :: Initialize a runtime stack
 */
EXTERN_C void emlrtHandleParallelRunTimeError(void);

/*
 * MATLAB INTERNAL USE ONLY :: Initialize a runtime stack
 */
EXTERN_C void emlrtHandleParallelSuppressedWarning(void);

/*
 * MATLAB INTERNAL USE ONLY :: Initialize a runtime stack
 */
EXTERN_C void emlrtEnterRtStackR2011b(struct emlrtContext *aContext, int32_T aCores);

/*
 * MATLAB INTERNAL USE ONLY :: Initialize a runtime stack
 */
EXTERN_C void emlrtEnterRtStack(struct emlrtContext *aContext);

/*
 * MATLAB INTERNAL USE ONLY :: Terminate a runtime stack
 */
EXTERN_C void emlrtLeaveRtStack(struct emlrtContext *aContext);

#define EMLRTPUSHRTSTACKR2011B(aRSInfo, aTId) { \
 if (emlrtContextGlobal.fRTCallStack->fRTStackPointer[aTId] < emlrtContextGlobal.fRTCallStack->fRTStackSize[aTId]) \
(emlrtContextGlobal.fRTCallStack->fRTStackInfo[aTId][emlrtContextGlobal.fRTCallStack->fRTStackPointer[aTId]++] = aRSInfo); \
else emlrtPushRtStackR2011b(aRSInfo,aTId); }

#define EMLRTPUSHRTSTACK(aRSInfo) { \
    if (emlrtContextGlobal.fRTCallStack->fRTStackPointer[0] < emlrtContextGlobal.fRTCallStack->fRTStackSize[0]) \
    (emlrtContextGlobal.fRTCallStack->fRTStackInfo[0][emlrtContextGlobal.fRTCallStack->fRTStackPointer[0]++] = aRSInfo); \
    else emlrtPushRtStack(aRSInfo); }

/*
 * MATLAB INTERNAL USE ONLY :: Push to runtime stack
 */
EXTERN_C void emlrtPushRtStackR2011b(const struct emlrtRSInfo *aRSInfo, int32_T aTId);

/*
 * MATLAB INTERNAL USE ONLY :: Push to runtime stack
 */
EXTERN_C void emlrtPushRtStack(const struct emlrtRSInfo *aRSInfo);

#define EMLRTPOPRTSTACKR2011B(aRSInfo, aTId) { \
    if (emlrtContextGlobal.fRTCallStack->fRTStackPointer[aTId] != 0) \
    (emlrtContextGlobal.fRTCallStack->fRTStackPointer[aTId]--); \
    else emlrtPopRtStackR2011b(aRSInfo,aTId); }

#define EMLRTPOPRTSTACK(aRSInfo) { \
    if (emlrtContextGlobal.fRTCallStack->fRTStackPointer[0] != 0) \
    (emlrtContextGlobal.fRTCallStack->fRTStackPointer[0]--); \
    else emlrtPopRtStack(aRSInfo); }

/*
 * MATLAB INTERNAL USE ONLY :: Pop from runtime stack
 */
EXTERN_C void emlrtPopRtStackR2011b(const struct emlrtRSInfo *aRSInfo, int32_T aTId);

/*
 * MATLAB INTERNAL USE ONLY :: Pop from runtime stack
 */
EXTERN_C void emlrtPopRtStack(const struct emlrtRSInfo *aRSInfo);

/*
 * MATLAB INTERNAL USE ONLY :: Serialize a byte
 */
EXTERN_C void
emlrtSerializeByte(uint8_T b);

/*
 * MATLAB INTERNAL USE ONLY :: Deserialize a byte
 */
EXTERN_C uint8_T
emlrtDeserializeByte(void);

/*
 * MATLAB INTERNAL USE ONLY :: Terminate serializing
 */
EXTERN_C void
emlrtSerializeTerminate(void);

/*
 * MATLAB INTERNAL USE ONLY :: Deserialize a double
 */
EXTERN_C real64_T
emlrtDeserializeDouble(void);

/*
 * MATLAB INTERNAL USE ONLY :: Serialize a double
 */
EXTERN_C void
emlrtSerializeDouble(real64_T d);

/*
 * MATLAB INTERNAL USE ONLY :: Deserialize a single
 */
EXTERN_C real32_T
emlrtDeserializeSingle(void);

/*
 * MATLAB INTERNAL USE ONLY :: Serialize a single
 */
EXTERN_C void
emlrtSerializeSingle(real32_T d);

/*
 * MATLAB INTERNAL USE ONLY :: Deserialize a char
 */
EXTERN_C char
emlrtDeserializeChar(void);

/*
 * MATLAB INTERNAL USE ONLY :: Serialize a char
 */
EXTERN_C void
emlrtSerializeChar(char c);

/*
 * MATLAB INTERNAL USE ONLY :: Deserialize a logical
 */
EXTERN_C boolean_T
emlrtDeserializeLogical(void);

/*
 * MATLAB INTERNAL USE ONLY :: Serialize a logical
 */
EXTERN_C void
emlrtSerializeLogical(boolean_T b);

/*
 * MATLAB INTERNAL USE ONLY :: Initialize serializing
 */
EXTERN_C void
emlrtSerializeInitialize(boolean_T isDeserialize, boolean_T isVerification, const char *projectName, uint32_T aCheckSumLen, const uint32_T *aChecksum);

#ifdef __WATCOMC__
#pragma aux emlrtDeserializeDouble value [8087];
#pragma aux emlrtDeserializeSingle value [8087];
#endif

/*
 * MATLAB INTERNAL USE ONLY :: Check for Ctrl+C (break)
 */
EXTERN_C void
emlrtBreakCheck(void);

/*
 * MATLAB INTERNAL USE ONLY :: Check for Ctrl+C (break)
 */
EXTERN_C void
emlrtBreakCheckR2011b(struct emlrtContext *aContext, int32_T aTId);

/*
 * MATLAB INTERNAL USE ONLY :: Equality check for 1-D sizes
 */
EXTERN_C void
emlrtSizeEqCheck1D(int32_T dim1, int32_T dim2, emlrtECInfo *aInfo);

/*
 * MATLAB INTERNAL USE ONLY :: Equality check for 1-D sizes
 */
EXTERN_C void
emlrtSizeEqCheck1DR2011a(int32_T dim1, int32_T dim2, emlrtECInfo *aInfo, struct emlrtContext *aContext);

/*
 * MATLAB INTERNAL USE ONLY :: Equality check for 1-D sizes
 */
EXTERN_C void
emlrtSizeEqCheck1DR2011b(int32_T dim1, int32_T dim2, emlrtECInfo *aInfo, struct emlrtContext *aContext, int32_T aTId);

/*
 * MATLAB INTERNAL USE ONLY :: Equality check for size vectors
 */
EXTERN_C void
emlrtSizeEqCheckND(const int32_T* dims1, const int32_T* dims2, emlrtECInfo *aInfo);

/*
 * MATLAB INTERNAL USE ONLY :: Equality check for size vectors
 */
EXTERN_C void
emlrtSizeEqCheckNDR2011a(const int32_T* dims1, const int32_T* dims2, emlrtECInfo *aInfo, struct emlrtContext *aContext);

/*
 * MATLAB INTERNAL USE ONLY :: Equality check for size vectors
 */
EXTERN_C void
emlrtSizeEqCheckNDR2011b(const int32_T* dims1, const int32_T* dims2, emlrtECInfo *aInfo, struct emlrtContext *aContext, int32_T aTId);

/*
 * MATLAB INTERNAL USE ONLY :: equality check
 */
EXTERN_C void
emlrtDimSizeEqCheck(int32_T dim1, int32_T dim2, emlrtECInfo *aInfo);

/*
 * MATLAB INTERNAL USE ONLY :: equality check
 */
EXTERN_C void
emlrtDimSizeEqCheckR2011a(int32_T dim1, int32_T dim2, emlrtECInfo *aInfo, struct emlrtContext *aContext);

/*
 * MATLAB INTERNAL USE ONLY :: equality check
 */
EXTERN_C void
emlrtDimSizeEqCheckR2011b(int32_T dim1, int32_T dim2, emlrtECInfo *aInfo, struct emlrtContext *aContext, int32_T aTId);

/*
 * MATLAB INTERNAL USE ONLY :: greater than or euqal to check
 */
EXTERN_C void
emlrtDimSizeGeqCheck(int32_T dim1, int32_T dim2, emlrtECInfo *aInfo);

/*
 * MATLAB INTERNAL USE ONLY :: greater than or euqal to check
 */
EXTERN_C void
emlrtDimSizeGeqCheckR2011a(int32_T dim1, int32_T dim2, emlrtECInfo *aInfo, struct emlrtContext *aContext);

/*
 * MATLAB INTERNAL USE ONLY :: greater than or euqal to check
 */
EXTERN_C void
emlrtDimSizeGeqCheckR2011b(int32_T dim1, int32_T dim2, emlrtECInfo *aInfo, struct emlrtContext *aContext, int32_T aTId);

/*
 * MATLAB INTERNAL USE ONLY :: Check size compatibility for A(I1,..IN) = B assignment in MATLAB.
 */
EXTERN_C void
emlrtSubAssignSizeCheck(const int32_T* dims1, int32_T nDims1, const int32_T* dims2, int32_T nDims2, emlrtECInfo *aInfo);

/*
 * MATLAB INTERNAL USE ONLY :: Check size compatibility for A(I1,..IN) = B assignment in MATLAB.
 */
EXTERN_C void
emlrtSubAssignSizeCheckR2011a(const int32_T* dims1, int32_T nDims1, const int32_T* dims2, int32_T nDims2, emlrtECInfo *aInfo, struct emlrtContext *aContext);

/*
 * MATLAB INTERNAL USE ONLY :: Check size compatibility for A(I1,..IN) = B assignment in MATLAB.
 */
EXTERN_C void
emlrtSubAssignSizeCheckR2011b(const int32_T* dims1, int32_T nDims1, const int32_T* dims2, int32_T nDims2, emlrtECInfo *aInfo, struct emlrtContext *aContext, int32_T aTId);

/*
 * MATLAB INTERNAL USE ONLY :: Check that at least one of the two given size vectors describe a proper
 * matrix (not a vector).
 */
EXTERN_C void emlrtMatrixMatrixIndexCheck(const int32_T* dims1, int32_T nDims1, const int32_T* dims2, int32_T nDims2, emlrtECInfo *aInfo);

/*
 * MATLAB INTERNAL USE ONLY :: Check that at least one of the two given size vectors describe a proper
 * matrix (not a vector).
 */
EXTERN_C void emlrtMatrixMatrixIndexCheckR2011a(const int32_T* dims1, int32_T nDims1, const int32_T* dims2, int32_T nDims2, emlrtECInfo *aInfo, struct emlrtContext *aContext);

/*
 * MATLAB INTERNAL USE ONLY :: Check that at least one of the two given size vectors describe a proper
 * matrix (not a vector).
 */
EXTERN_C void emlrtMatrixMatrixIndexCheckR2011b(const int32_T* dims1, int32_T nDims1, const int32_T* dims2, int32_T nDims2, emlrtECInfo *aInfo, struct emlrtContext *aContext, int32_T aTId);

/*
 * MATLAB INTERNAL USE ONLY :: Check that at least one of the two given size vectors describe a proper
 * matrix (not a vector).
 */
EXTERN_C void emlrtVectorVectorIndexCheck(int32_T sizeL_0, int32_T sizeL_1, int32_T sizeR_0, int32_T sizeR_1, emlrtECInfo *aInfo);

/*
 * MATLAB INTERNAL USE ONLY :: Check that at least one of the two given size vectors describe a proper
 * matrix (not a vector).
 */
EXTERN_C void emlrtVectorVectorIndexCheckR2011a(int32_T sizeL_0, int32_T sizeL_1, int32_T sizeR_0, int32_T sizeR_1, emlrtECInfo *aInfo, struct emlrtContext *aContext);

/*
 * MATLAB INTERNAL USE ONLY :: Check that at least one of the two given size vectors describe a proper
 * matrix (not a vector).
 */
EXTERN_C void emlrtVectorVectorIndexCheckR2011b(int32_T sizeL_0, int32_T sizeL_1, int32_T sizeR_0, int32_T sizeR_1, emlrtECInfo *aInfo, struct emlrtContext *aContext, int32_T aTId);

EXTERN_C char *
emlrtExtractMessageId(const struct emlrtMsgIdentifier *aMsgId);

/*
 * MATLAB INTERNAL USE ONLY :: Return true if this is an MCOS enumeration.
 */
EXTERN_C bool
emlrtIsEnumR2009a(const mxArray *mx);

/*
 * MATLAB INTERNAL USE ONLY :: Check the class of an mxArray
 */
EXTERN_C void
emlrtCheckClass(const char *msgName, const mxArray *pa, const char *className);

/*
 * MATLAB INTERNAL USE ONLY :: Check the sparseness of an mxArray
 */
EXTERN_C void
emlrtCheckSparse(const char *msgName, const mxArray *pa, boolean_T sparse);

/*
 * MATLAB INTERNAL USE ONLY :: Check the size, class and complexness of an mxArray
 */
EXTERN_C void
emlrtCheckBuiltInR2011a(const struct emlrtMsgIdentifier *aMsgId, const mxArray *pa,
                  const char *className, boolean_T complex, uint32_T nDims, const void *pDims);

/*
 * MATLAB INTERNAL USE ONLY :: Check the size, class and complexness of an mxArray
 */
EXTERN_C void
emlrtCheckBuiltInCtxR2011b(emlrtContext *aCtx,
                           const struct emlrtMsgIdentifier *aMsgId, const mxArray *pa,
                           const char *className, boolean_T complex, uint32_T nDims, const void *pDims);

/*
 * MATLAB INTERNAL USE ONLY :: Check the size, class and complexness of an mxArray
 */
EXTERN_C void
emlrtCheckBuiltInCtxR2011a(struct emlrtContext *aCtx,
                           const struct emlrtMsgIdentifier *aMsgId, const mxArray *pa,
                           const char *className, boolean_T complex, uint32_T nDims, const void *pDims);

/*
 * MATLAB INTERNAL USE ONLY :: Check the size, class and complexness of an mxArray
 */
EXTERN_C void
emlrtCheckBuiltIn(const char *msgName, const mxArray *pa,
                  const char *className, boolean_T complex, uint32_T nDims, const void *pDims);

/*
 * MATLAB INTERNAL USE ONLY :: Check the size, class and complexness of an mxArray
 */
EXTERN_C void
emlrtCheckBuiltInR2009a(struct emlrtContext *aCtx,
                        const char *msgName, const mxArray *pa,
                        const char *className, boolean_T complex, uint32_T nDims, const void *pDims);

/*
 * MATLAB INTERNAL USE ONLY :: Check the size, class and complexness of a variable-size mxArray
 */
EXTERN_C void
emlrtCheckVsBuiltInR2011a(const struct emlrtMsgIdentifier *aMsgId, const mxArray *pa,
                    const char *className, boolean_T complex, uint32_T nDims, const void *pDims,
                    const boolean_T *aDynamic, int32_T *aOutSizes);

/*
 * MATLAB INTERNAL USE ONLY :: Check the size, class and complexness of a variable-size mxArray
 */
EXTERN_C void
emlrtCheckVsBuiltInCtxR2011b(struct emlrtContext *aCtx,
                             const struct emlrtMsgIdentifier *aMsgId, const mxArray *pa,
                             const char *className, boolean_T complex, uint32_T nDims, const void *pDims,
                             const boolean_T *aDynamic, int32_T *aOutSizes);

/*
 * MATLAB INTERNAL USE ONLY :: Check the size, class and complexness of a variable-size mxArray
 */
EXTERN_C void
emlrtCheckVsBuiltInR2008b(const char *msgName, const mxArray *pa,
                    const char *className, boolean_T complex, uint32_T nDims, const void *pDims,
                    const boolean_T *aDynamic, int32_T *aOutSizes);

/*
 * MATLAB INTERNAL USE ONLY :: Check the size, class and complexness of a variable-size mxArray
 */
EXTERN_C void
emlrtCheckVsBuiltInR2009a(emlrtContext *aCtx,
                          const char *msgName, const mxArray *pa,
                          const char *className, boolean_T complex, uint32_T nDims, const void *pDims,
                          const boolean_T *aDynamic, int32_T *aOutSizes);

/*
 * MATLAB INTERNAL USE ONLY :: Check the size, class and complexness of a variable-size mxArray
 */
EXTERN_C void
emlrtCheckVsBuiltInCtxR2011a(emlrtContext *aCtx,
                          const struct emlrtMsgIdentifier *aMsgId, const mxArray *pa,
                          const char *className, boolean_T complex, uint32_T nDims, const void *pDims,
                          const boolean_T *aDynamic, int32_T *aOutSizes);

/*
 * MATLAB INTERNAL USE ONLY :: Check the type of a FI mxArray
 */
EXTERN_C void
emlrtCheckFiR2011a(const struct emlrtMsgIdentifier *aMsgId, const mxArray *aFi, boolean_T aComplex, uint32_T aNDims, const void *aVDims,
             const mxArray *aFimath, const mxArray *aNumericType);

/*
 * MATLAB INTERNAL USE ONLY :: Check the type of a FI mxArray
 */
EXTERN_C void
emlrtCheckFiCtxR2011b(emlrtContext *aCtx,
                      const struct emlrtMsgIdentifier *aMsgId, const mxArray *aFi, boolean_T aComplex,
                      uint32_T aNDims, const void *aVDims,
                      const mxArray *aFimath, const mxArray *aNumericType);

/*
 * MATLAB INTERNAL USE ONLY :: Check the type of a FI mxArray
 */
EXTERN_C void
emlrtCheckFI(const char *aMsgName, const mxArray *aFi, boolean_T aComplex, uint32_T aNDims, const void *aVDims,
             const mxArray *aFimath, const mxArray *aNumericType);

/*
 * MATLAB INTERNAL USE ONLY :: Check the type of a variable-size FI mxArray
 */
EXTERN_C void
emlrtCheckVsFiR2011a(const struct emlrtMsgIdentifier *aMsgId, const mxArray *aFi, boolean_T aComplex, uint32_T aNDims, const void *aVDims,
                     const boolean_T *aDynamic, const mxArray *aFimath, const mxArray *aNumericType);

/*
 * MATLAB INTERNAL USE ONLY :: Check the type of a variable-size FI mxArray
 */
EXTERN_C void
emlrtCheckVsFiCtxR2011b(emlrtContext *aCtx,
                        const struct emlrtMsgIdentifier *aMsgId, const mxArray *aFi, boolean_T aComplex,
                        uint32_T aNDims, const void *aVDims,
                        const boolean_T *aDynamic, const mxArray *aFimath, const mxArray *aNumericType);

/*
 * MATLAB INTERNAL USE ONLY :: Check the type of a variable-size FI mxArray
 */
EXTERN_C void
emlrtCheckVsFiR2010b(const char *aMsgName, const mxArray *aFi, boolean_T aComplex, uint32_T aNDims, const void *aVDims,
                     const boolean_T *aDynamic, const mxArray *aFimath, const mxArray *aNumericType);

/*
 * MATLAB INTERNAL USE ONLY :: Check the type of a variable-size FI mxArray
 */
EXTERN_C void
emlrtCheckVsFiR2008b(const char *aMsgName, const mxArray *aFi, boolean_T aComplex, uint32_T aNDims, const void *aVDims,
                     const boolean_T *aDynamic, int32_T *aOutSizes,
                     const mxArray *aFimath, const mxArray *aNumericType);

/*
 * MATLAB INTERNAL USE ONLY :: Check the type of a static-size struct mxArray
 */
EXTERN_C void
emlrtCheckStructR2011a(const emlrtMsgIdentifier *aMsgId, const mxArray *s, int32_T nFields, const char **fldNames,
                 uint32_T nDims, const void *pDims);

/*
 * MATLAB INTERNAL USE ONLY :: Check the type of a static-size struct mxArray
 */
EXTERN_C void
emlrtCheckStruct(const char *msgName, const mxArray *s, int32_T nFields, const char **fldNames,
                 uint32_T nDims, const void *pDims);

/*
 * MATLAB INTERNAL USE ONLY :: Check the type of a variable-size struct mxArray
 */
EXTERN_C void
emlrtCheckVsStructR2011a(const struct emlrtMsgIdentifier *aMsgId, const mxArray *s, int32_T nFields, const char **fldNames,
                   uint32_T nDims, const void *pDims,
                   const boolean_T *aDynamic, int32_T *aOutSizes);

/*
 * MATLAB INTERNAL USE ONLY :: Check the type of a variable-size struct mxArray
 */
EXTERN_C void
emlrtCheckVsStructR2008b(const char *msgName, const mxArray *s, int32_T nFields, const char **fldNames,
                   uint32_T nDims, const void *pDims,
                   const boolean_T *aDynamic, int32_T *aOutSizes);

/*
 * MATLAB INTERNAL USE ONLY :: Check the type of a static-size struct mxArray
 */
EXTERN_C void
emlrtCheckEnumR2009a(emlrtContext *aCtx, const char *enumName, int32_T nEnumElements, const char **enumNames, const int32_T *enumValues);

/*
 * MATLAB INTERNAL USE ONLY :: Check the type of an unused input
 */
EXTERN_C void
emlrtCheckUnusedR2009b(void *aUnused, size_t aSize);

/*
 * MATLAB INTERNAL USE ONLY :: Import a character array.
 */
EXTERN_C void
emlrtImportCharArray(const mxArray *aSrc, char_T *aDst, int32_T aNumel);

/*
 * MATLAB INTERNAL USE ONLY :: Import a character.
 */
EXTERN_C void
emlrtImportChar(const mxArray *aSrc, char_T *aDst);

/*
 * MATLAB INTERNAL USE ONLY :: Set the actual size of a variable-size array
 */
extern void
emlrtSetVsSizesR2008b(const mxArray *pa, uint32_T nDimsMax, int32_T *aOutSizes);

/*
 * MATLAB INTERNAL USE ONLY :: Import an mxArray
 */
EXTERN_C void
emlrtImportArrayR2008b(const mxArray *aIn, void *aOutData, int32_T aElementSize);

/*
 * MATLAB INTERNAL USE ONLY :: Import an mxArray
 */
EXTERN_C void
emlrtImportArrayR2011b(const mxArray *aIn, void *aOutData, int32_T aElementSize, boolean_T aComplex);

/*
 * MATLAB INTERNAL USE ONLY :: Import an mxArray
 */
EXTERN_C void
emlrtImportVsArrayR2008b(const mxArray *aIn, void *aOutData, int32_T aElementSize, uint32_T nDimsMax, int32_T *aOutSizes);

/*
 * MATLAB INTERNAL USE ONLY :: Import a FI mxArray
 */
EXTERN_C void
emlrtImportVsFiArrayR2011b(const mxArray *aFiMx, const mxArray *aIntMx, void *aOutData, int32_T aElementSize, boolean_T aComplex, uint32_T nDimsMax, int32_T *aOutSizes);

/*
 * MATLAB INTERNAL USE ONLY :: Import a FI mxArray
 */
EXTERN_C void
emlrtImportVsFiArrayR2009b(const mxArray *aFiMx, const mxArray *aIntMx, void *aOutData, int32_T aElementSize, uint32_T nDimsMax, int32_T *aOutSizes);

/*
 * MATLAB INTERNAL USE ONLY :: Set the actual sizes of a dynamic FI array
 */
EXTERN_C void
emlrtSetVsFiSizes(const mxArray *aFi, uint32_T nDimsExpected, int32_T *aOutSizes);

#endif /* emlrt_h */
```

### engine.h
```c
/*
 * @(#)engine.h    generated by: makeheader 5.1.5  Tue May 24 21:08:29 2011
 *
 *		built from:	../../src/include/copyright.h
 *				../../src/include/pragma_interface.h
 *				engapi.cpp
 *				fengapi.cpp
 */

#if defined(_MSC_VER)
# pragma once
#endif
#if defined(__GNUC__) && (__GNUC__ > 3 || (__GNUC__ == 3 && __GNUC_MINOR__ > 3))
# pragma once
#endif

#ifndef engine_h
#define engine_h

/*
 * Copyright 1984-2003 The MathWorks, Inc.
 * All Rights Reserved.
 */

/* Copyright 2003-2006 The MathWorks, Inc. */

/* Only define EXTERN_C if it hasn't been defined already. This allows
 * individual modules to have more control over managing their exports.
 */
#ifndef EXTERN_C

#ifdef __cplusplus
  #define EXTERN_C extern "C"
#else
  #define EXTERN_C extern
#endif

#endif

#include "matrix.h"     /* mx Routines used in module */

typedef struct engine Engine;	/* Incomplete definition for Engine */

/*
 * Execute matlab statement
 */
EXTERN_C int engEvalString(
	Engine	*ep,		/* engine pointer */
	const char *string	/* string for matlab t execute */
	);

/*
 * Start matlab process for single use.
 * Not currently supported on UNIX.
 */
EXTERN_C Engine *engOpenSingleUse(
			 const char *startcmd, /* exec command string used to start matlab */
			 void *reserved, /* reserved for future use, must be NULL */
			 int *retstatus /* return status */
);

/*
 * SetVisible, do nothing since this function is only for NT
 */
EXTERN_C int engSetVisible(
		  Engine *ep,        /* engine pointer */
		  bool newVal
		  );

/*
 * GetVisible, do nothing since this function is only for NT
 */
EXTERN_C int engGetVisible(
		  Engine *ep,        /* engine pointer */
		  bool* bVal
		  );

/*
 * Start matlab process
 */
EXTERN_C Engine *engOpen(
	const char *startcmd /* exec command string used to start matlab */
	);

/*
 * Close down matlab server
 */
EXTERN_C int engClose(
	Engine	*ep         /* engine pointer */
	);

/*
 * Get a variable with the specified name from MATLAB's workspace
 */
EXTERN_C mxArray *engGetVariable(
	Engine	*ep,		/* engine pointer */
	const char *name	/* name of variable to get */
	);

/*
 * Put a variable into MATLAB's workspace with the specified name
 */
EXTERN_C int engPutVariable(
		   Engine	*ep,        /* engine pointer */
		   const char *var_name,
		   const mxArray *ap   /* array pointer */
		   );

/*
 * register a buffer to hold matlab text output
 */
EXTERN_C int engOutputBuffer(
	Engine	*ep,		/* engine pointer */
	char	*buffer,	/* character array to hold output */
	int     buflen		/* buffer array length */
	);

#endif /* engine_h */
```

### ext_share.h
```c
/* File: ext_share.h
 * Absract:
 *	External mode shared data structures used by the external communication
 *	mex link, the generated code, and Simulink.
 *
 * Copyright 1994-2005 The MathWorks, Inc.
 *
 * $Revision: 1.14.4.6 $
 */

#ifndef __EXTSHARE__
#define __EXTSHARE__

typedef enum {
    /*================================
     * Packets/actions to target.
     *==============================*/

    /* connection actions */
    EXT_CONNECT,
    EXT_DISCONNECT_REQUEST,
    EXT_DISCONNECT_REQUEST_NO_FINAL_UPLOAD,
    EXT_DISCONNECT_CONFIRMED,

    /* parameter upload/download actions */
    EXT_SETPARAM,
    EXT_GETPARAMS,

    /* data upload actions */
    EXT_SELECT_SIGNALS,
    EXT_SELECT_TRIGGER,
    EXT_ARM_TRIGGER,
    EXT_CANCEL_LOGGING,

    /* model control actions */
    EXT_MODEL_START,
    EXT_MODEL_STOP,
    EXT_MODEL_PAUSE,
    EXT_MODEL_STEP,
    EXT_MODEL_CONTINUE,

    /* data request actions */
    EXT_GET_TIME,

    /*================================
     * Packets/actions from target.
     *==============================*/

    /* responses */
    EXT_CONNECT_RESPONSE,   /* must not be 0! */
    EXT_DISCONNECT_REQUEST_RESPONSE,
    EXT_SETPARAM_RESPONSE,
    EXT_GETPARAMS_RESPONSE,
    EXT_MODEL_SHUTDOWN,
    EXT_GET_TIME_RESPONSE,
    EXT_MODEL_START_RESPONSE,
    EXT_MODEL_PAUSE_RESPONSE,
    EXT_MODEL_STEP_RESPONSE,
    EXT_MODEL_CONTINUE_RESPONSE,
    EXT_UPLOAD_LOGGING_DATA,
    EXT_SELECT_SIGNALS_RESPONSE,
    EXT_SELECT_TRIGGER_RESPONSE,
    EXT_ARM_TRIGGER_RESPONSE,
    EXT_CANCEL_LOGGING_RESPONSE,

    /*
     * This packet is sent from the target to signal the end of a data
     * collection event (e.g., each time that the duration is reached).
     * This packet only applies to normal mode (see
     * EXT_TERMINATE_LOG_SESSION)
     */
    EXT_TERMINATE_LOG_EVENT,

    /*
     * This packet is sent from the target at the end of each data logging
     * session.  This occurs either at the end of a oneshot or at the end
     * of normal mode (i.e., the last in a series of oneshots).
     */
    EXT_TERMINATE_LOG_SESSION,

    EXTENDED = 255          /* reserved for extending beyond 254 ID's */
} ExtModeAction;

typedef enum {
  STATUS_OK,
  NOT_ENOUGH_MEMORY
} ResponseStatus;

typedef enum {
  LittleEndian,
  BigEndian
} MachByteOrder;

#ifndef TARGETSIMSTATUS_DEFINED
#define TARGETSIMSTATUS_DEFINED
typedef enum {
    TARGET_STATUS_NOT_CONNECTED,
    TARGET_STATUS_WAITING_TO_START,
    TARGET_STATUS_STARTING, /* in the process of starting - host waiting
                               for confirmation */

    TARGET_STATUS_RUNNING,
    TARGET_STATUS_PAUSED
} TargetSimStatus;
#endif

/*
 * The packet header consists of 2 32 bit unsigned ints [type, size].  size
 * is the number of bytes coming after the header.  It is always expressed
 * in target bytes.
 */
typedef struct PktHeader_tag {
    uint32_T type;  /* packet type */
    uint32_T size;  /* number of bytes to follow */
} PktHeader;
#define NUM_HDR_ELS (2)

#ifndef FALSE
enum {FALSE, TRUE};
#endif

#define NO_ERR (0)

#define EXT_NO_ERROR ((boolean_T)(0))
#define EXT_ERROR ((boolean_T)(1))

#define UNKNOWN_BYTES_NEEDED (-1)

#define PRIVATE static
#define PUBLIC

#endif /* __EXTSHARE__ */
```

### ext_svr.h
```c
/*
 * Copyright 1994-2008 The MathWorks, Inc.
 *
 * File: ext_svr.h     $Revision: 1.1.6.6 $
 *
 * Abstract:
 *	Function prototypes for provided TCP socket based external mode
 *      implementation.
 */

#ifndef __EXT_SVR__
#define __EXT_SVR__

#include "ext_share.h"

#ifdef __cplusplus

extern "C" {

#endif

extern boolean_T SendPktToHost(const ExtModeAction action,
                               const int           size,
                               const char          *data);

extern boolean_T rt_ExtModeInit(void);

extern void      rt_PktServerWork(RTWExtModeInfo *ei,
                                  int_T          numSampTimes,
                                  boolean_T      *stopReq);

extern void      rt_UploadServerWork(int_T numSampTimes);

extern boolean_T rt_ExtModeShutdown(int_T numSampTimes);

extern void      rt_UploadCheckTrigger(int_T numSampTimes);

extern void      rt_UploadCheckEndTrigger(void);

extern void      rt_UploadBufAddTimePoint(int_T tid,
                                          real_T taskTime);

#ifndef VXWORKS
extern void      rt_ExtModeSleep(long sec,   /* number of seconds to wait      */
                                 long usec); /* number of micro seconds to wait*/
#else
extern void      rt_UploadServer(int_T numSampTimes);

extern void      rt_PktServer(RTWExtModeInfo *ei,
                              int_T          numSampTimes,
                              boolean_T      *stopReq);

extern void      rt_SetPortInExtUD(const int_T port);
#endif

extern const char_T *ExtParseArgsAndInitUD(const int_T  argc,
                                           const char_T *argv[]);
extern boolean_T  ExtWaitForStartPkt(void);

#ifdef __cplusplus

}
#endif

#endif /* __EXT_SVR__ */

/* [EOF] ext_svr.h */
```

### ext_svr_transport.h
```c
/*
 * Copyright 1994-2002 The MathWorks, Inc.
 *
 * File: ext_svr_transport.h     $Revision: 1.1.6.1 $
 *
 * Abstract:
 *  PUBLIC interface for ext_svr_transport.c.
 */

/********************* DO NOT CHANGE BELOW THIS LINE **************************
 *                                                                            *
 * The function prototypes below define the interface between the target-     *
 * side external mode and ext_svr_transport.  They should not need to be      *
 * changed.  Only the implementation of these functions in ext_svr_transport.c*
 * should need to be modified.                                                *
 *                                                                            *
 ******************************************************************************/

/*
 * Export the user data as an 'opaque' or 'incomplete' data type.  ext_svr
 * may reference it (i.e., pass pointers to it, but it can not dereference
 * the pointer).
 */
typedef struct ExtUserData_tag ExtUserData;

/*
 * Define the transport interface.
 */

extern boolean_T ExtInit(ExtUserData *UD);

extern boolean_T ExtOpenConnection(
    ExtUserData *UD,
    boolean_T   *outConnectionMade);

extern void ExtCloseConnection(ExtUserData *UD);

extern void ExtShutDown(ExtUserData *UD);

extern const char_T *ExtProcessArgs(
    ExtUserData   *UD,
    const int_T   argc,
    const char_T  *argv[]);

extern boolean_T ExtWaitForStartPktFromHost(ExtUserData *UD);

extern ExtUserData *ExtUserDataCreate(void);

extern void ExtUserDataDestroy(ExtUserData *userData);

#ifdef VXWORKS
extern void ExtUserDataSetPort(ExtUserData *UD, const int_T port);
#endif

extern boolean_T ExtGetHostPkt(
    const ExtUserData *UD,
    const int         nBytesToGet,
    int               *nBytesGot,
    char              *dst);

extern boolean_T ExtSetHostPkt(
    const ExtUserData *UD,
    const int         nBytesToSet,
    const char        *src,
    int               *nBytesSet);

extern void ExtModeSleep(
    const ExtUserData *UD,
    const long        sec,
    const long        usec);

extern void ExtForceDisconnect(ExtUserData *UD);
```

### ext_test.h
```c
/*
 * Copyright 1994-2002 The MathWorks, Inc.
 *
 * File: ext_test.h     $Revision: 1.1.6.1 $
 *
 * Abstract:
 *
 */

#ifndef __EXT_TEST_OBJECT__
#define __EXT_TEST_OBJECT__

#ifdef TMW_EXTMODE_TESTING
extern void rtExtModeTestingInit(void);
extern void rtExtModeTestingKillIfOrphaned(boolean_T pktReceived);
extern void rtExtModeTestingRemoveBatMarker(void);
#else
#define rtExtModeTestingInit()                      /* do nothing */
#define rtExtModeTestingKillIfOrphaned(pktReceived) /* do nothing */
#define rtExtModeTestingRemoveBatMarker()           /* do nothing */
#endif

#endif /* __EXT_TEST_OBJECT__ */
```

### ext_types.h
```c
/*
 * Copyright 1994-2004 The MathWorks, Inc.
 *
 * File: ext_types.h     $Revision: 1.1.6.3 $
 *
 * Abstract:
 */

#ifndef __EXT_TYPES__
#define __EXT_TYPES__

/* Additional types required for Simulink External Mode */
#ifndef fcn_call_T
# define fcn_call_T real_T
#endif
#ifndef action_T
# define action_T real_T
#endif

/****************************************
 * Dynamic vs. Static memory allocation *
 ****************************************/
#ifdef EXTMODE_STATIC
#  include "mem_mgr.h"
#  define malloc ExtModeMalloc
#  define calloc ExtModeCalloc
#  define free   ExtModeFree
#endif

/****************************************
 * Integer only code                    *
 ****************************************/
#ifdef EXT_MODE
#  if INTEGER_CODE == 1
#    undef  real_T
#    define real_T int32_T

#    undef  real32_T
#    define real32_T int32_T

#    undef  double
#    define double int32_T

#    undef  time_T
#    define time_T int32_T
#  endif /* INTEGER_CODE == 1 */
#endif /* #ifdef EXTMODE */

#endif /* __EXT_TYPES__ */

/* [EOF] ext_types.h */
```

### ext_work.h
```c
/*
 * Copyright 1994-2005 The MathWorks, Inc.
 *
 * File: ext_work.h     $Revision: 1.1.6.11 $
 *
 * Abstract:
 *
 */

#ifndef __EXT_WORK_OBJECT__
#define __EXT_WORK_OBJECT__

#ifdef __cplusplus
extern "C" {
#endif

#ifdef EXT_MODE
#include "ext_types.h"

#if defined(VXWORKS)
    /*VxWorks headers*/
    #include <vxWorks.h>
    #include <taskLib.h>
    #include <sysLib.h>
    #include <semLib.h>
    #include <rebootLib.h>
    #include <logLib.h>

    extern void rtExtModeTornadoStartup(RTWExtModeInfo *ei,
                                        int_T          numSampTimes,
                                        boolean_T      *stopReqPtr,
                                        int_T          priority,
                                        int32_T        stack_size,
                                        SEM_ID         startStopSem);

    extern void rtExtModeTornadoCleanup(int_T numSampTimes);

    extern void rtExtModeTornadoSetPortInExtUD(const int_T port);

#elif defined(C6000_EXT_MODE)
    /* C6000 headers*/
    #include <std.h>
    #include <stddef.h>
    #include <sem.h>

    extern void rtExtModeC6000Startup( RTWExtModeInfo *ei,
                                       int_T          numSampTimes,
                                       boolean_T      *stopReqPtr);

    extern void rtExtModeC6000Cleanup(int_T numSampTimes);
#else
    extern void rtExtModePauseIfNeeded(RTWExtModeInfo *ei,
                                       int_T          numSampTimes,
                                       boolean_T      *stopReqPtr);

    extern void rtExtModeWaitForStartPkt(RTWExtModeInfo *ei,
                                         int_T          numSampTimes,
                                         boolean_T      *stopReqPtr);
    void rtExtModeInitUD(void);
#endif /* #if defined(VXWORKS) */

extern void rtExtModeOneStep(RTWExtModeInfo *ei,
                             int_T          numSampTimes,
                             boolean_T      *stopReqPtr);

extern void rtExtModeCheckEndTrigger(void);

extern void rtExtModeUploadCheckTrigger(int_T numSampTimes);

extern void rtExtModeUpload(int_T tid,
                            real_T taskTime);

extern void rtExtModeCheckInit(int_T numSampTimes);

extern void rtExtModeShutdown(int_T numSampTimes);

extern void rtExtModeParseArgs(int_T        argc,
                               const char_T *argv[],
                               real_T       *rtmFinal);

extern void rtERTExtModeSetTFinal(real_T *rtmTFinal);

extern void rtERTExtModeParseArgs(int_T        argc,
                                  const char_T *argv[]);
extern void rtERTExtModeStartMsg(void);

#else /* #ifdef EXTMODE */

#if defined(VXWORKS)
    #define rtExtModeTornadoStartup(ei,                          \
                                    numSampTimes,                \
                                    stopReqPtr,                  \
                                    priority,                    \
                                    stack_size,                  \
                                    startStopSem) /* do nothing */
    #define rtExtModeTornadoCleanup(numSampTimes); /* do nothing */
    #define rtExtModeTornadoSetPortInExtUD(port); /* do nothing */
#elif defined(C6000_EXT_MODE)
    #define rtExtModePauseIfNeeded(ei,st,sr) /* do nothing */
    #define rtExtModeWaitForStartPkt(ei,st,sr) /* do nothing */
#else
    #define rtExtModePauseIfNeeded(ei,st,sr) /* do nothing */
    #define rtExtModeWaitForStartPkt(ei,st,sr) /* do nothing */
#endif /* #ifdef VXWORKS */

#define rtExtModeOneStep(ei,st,sr) /* do nothing */
#define rtExtModeCheckEndTrigger() /* do nothing */
#define rtExtModeUploadCheckTrigger(numSampTimes) /* do nothing */
#define rtExtModeUpload(t,ttime) /* do nothing */
#define rtExtModeCheckInit(numSampTimes) /* do nothing */
#define rtExtModeShutdown(numSampTimes) /* do nothing */
#define rtExtModeParseArgs(argc, argv, tf); /* do nothing */
#define rtERTExtModeSetTFinal(tf); /* do nothing */
#define rtERTExtModeParseArgs(argc, argv); /* do nothing */
#define rtERTExtModeStartMsg(); /* do nothing */

#endif  /* #ifdef EXTMODE */

#ifdef __cplusplus
}
#endif

#endif /* __EXT_WORK_OBJECT__ */
```
